// TIA Portal V17 export
// export: Created 2025-03-07T09:18:19.4347644Z, ExportSetting WithDefaults, DisplayName Totally Integrated Automation Portal, DisplayVersion V17 Update 8, DisplayName TIA Portal Openness, DisplayVersion V17 Update 8, DisplayName TIA Portal Version Control Interface, DisplayVersion V17, DisplayName SINAMICS Startdrive Advanced, DisplayVersion V17 SP2, DisplayName SINAMICS Startdrive G110M, G120, G120C, G120D, G120P, G115D, DisplayVersion V17 SP2, DisplayName SINAMICS Startdrive G130, G150, S120, S150, SINAMICS MV, S210, DisplayVersion V17 SP2, DisplayName STEP 7 Professional, DisplayVersion V17 Update 8, DisplayName SINUMERIK ONE STEP 7 Toolbox, DisplayVersion V17 Update 12, DisplayName SINUMERIK 840D sl STEP 7 Toolbox, DisplayVersion V17 Update 12, DisplayName STEP 7 Safety, DisplayVersion V17 Update 6, DisplayName WinCC Advanced, DisplayVersion V17 Update 8
FUNCTION "FC1702_ASPIRATION_VALVE" : Void   // FC1702, LAD
{ S7_Optimized_Access := 'TRUE' }
VERSION : 0.1
// stored: AutoNumber false, IsIECCheckEnabled false, SetENOAutomatically false, UDAEnableTagReadback false
BEGIN

REGION Network 1: <<<<<<<<<<<<<<<<<<<< ASPIRATION VALVES >>>>>>>>>>>>>>>>>>>>
END_REGION

REGION Network 2: <<<<<<<<<<<<<<<<<<<<<<<<<<< UNIT 01 >>>>>>>>>>>>>>>>>>>>>>>>>>>
END_REGION

REGION Network 3: CALL FB1701 UNIT 01 STATION 1 ASPIRATION ACTIVATION
   // 2#0000_0001 OPTIONS 0 BIT 0 SWITCHED ON INPUT 1 OPTION
   // 2#0000_0010 OPTIONS 0 BIT 1 SWITCHED ON INPUT 2 OPTION
   // 2#0000_0100 OPTIONS 0 BIT 2 SWITCHED ON INPUT 3 OPTION
   // 2#0000_1000 OPTIONS 0 BIT 3 SWITCHED ON INPUT 4 OPTION
   // 2#0001_0000 OPTIONS 0 BIT 4 SWITCHED OFF NOT SWITCHED ON INPUT 1 OPTION
   // 2#0010_0000 OPTIONS 0 BIT 5 SPARE
   // 2#0100_0000 OPTIONS 0 BIT 6 SPARE
   // 2#1000_0000 OPTIONS 0 BIT 7 SPARE
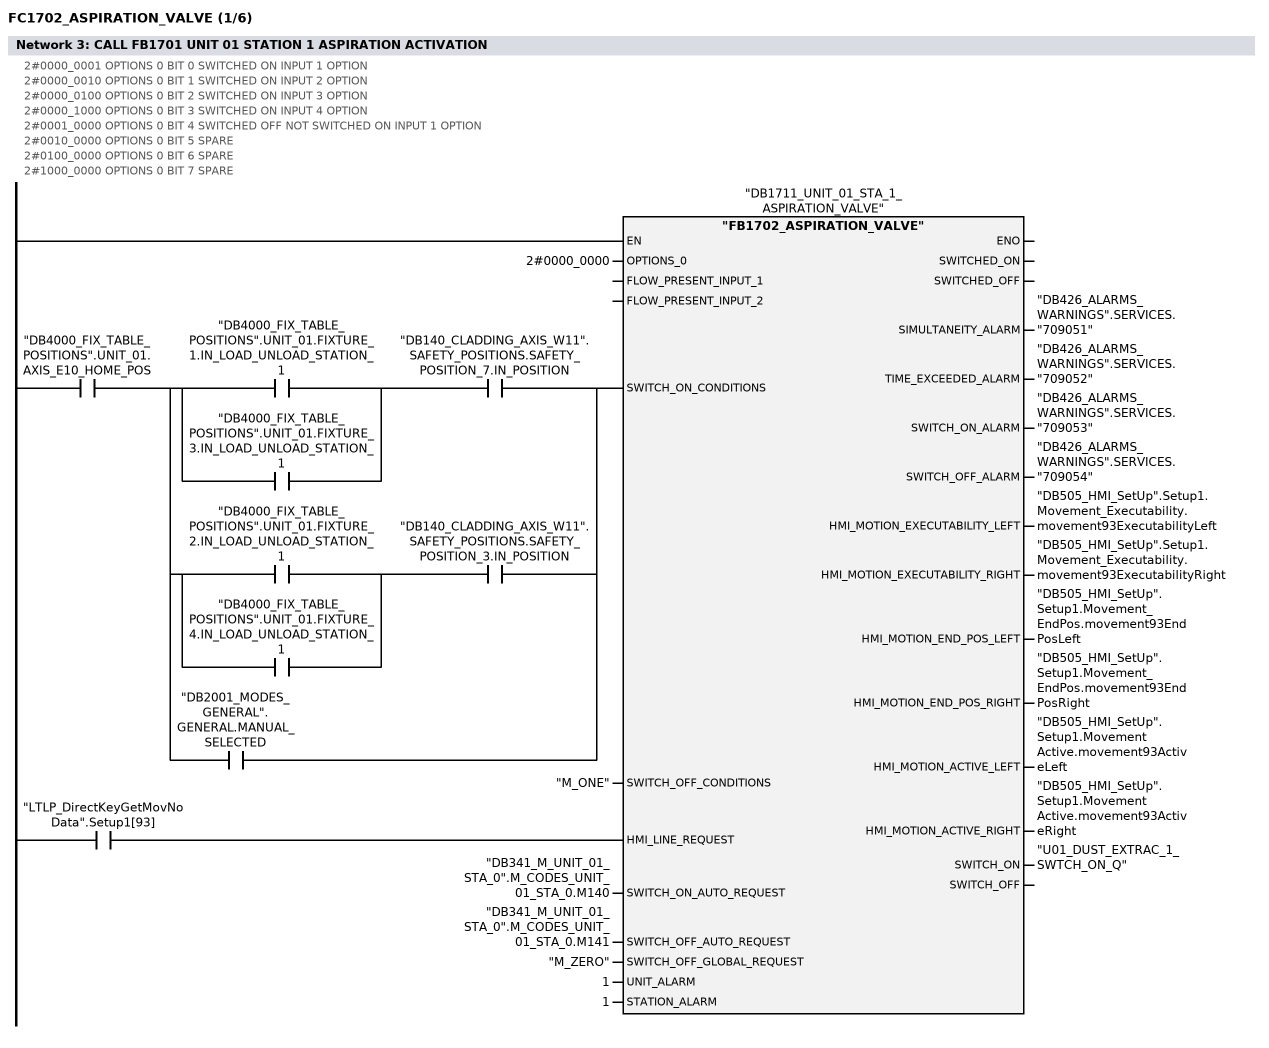
   RUNG wire#powerrail
      "DB1711_UNIT_01_STA_1_ASPIRATION_VALVE"(SWITCH_ON_CONDITIONS := wire#w4, HMI_LINE_REQUEST := wire#w5, OPTIONS_0 := 2#0000_0000, FLOW_PRESENT_INPUT_1 :=, FLOW_PRESENT_INPUT_2 :=, SWITCH_OFF_CONDITIONS := "M_ONE", SWITCH_ON_AUTO_REQUEST := "DB341_M_UNIT_01_STA_0".M_CODES_UNIT_01_STA_0.M140, SWITCH_OFF_AUTO_REQUEST := "DB341_M_UNIT_01_STA_0".M_CODES_UNIT_01_STA_0.M141, SWITCH_OFF_GLOBAL_REQUEST := "M_ZERO", UNIT_ALARM := 1, STATION_ALARM := 1, SWITCHED_ON =>, SWITCHED_OFF =>, SIMULTANEITY_ALARM => "DB426_ALARMS_WARNINGS".SERVICES."709051", TIME_EXCEEDED_ALARM => "DB426_ALARMS_WARNINGS".SERVICES."709052", SWITCH_ON_ALARM => "DB426_ALARMS_WARNINGS".SERVICES."709053", SWITCH_OFF_ALARM => "DB426_ALARMS_WARNINGS".SERVICES."709054", HMI_MOTION_EXECUTABILITY_LEFT => "DB505_HMI_SetUp".Setup1.Movement_Executability.movement93ExecutabilityLeft, HMI_MOTION_EXECUTABILITY_RIGHT => "DB505_HMI_SetUp".Setup1.Movement_Executability.movement93ExecutabilityRight, HMI_MOTION_END_POS_LEFT => "DB505_HMI_SetUp".Setup1.Movement_EndPos.movement93EndPosLeft, HMI_MOTION_END_POS_RIGHT => "DB505_HMI_SetUp".Setup1.Movement_EndPos.movement93EndPosRight, HMI_MOTION_ACTIVE_LEFT => "DB505_HMI_SetUp".Setup1.MovementActive.movement93ActiveLeft, HMI_MOTION_ACTIVE_RIGHT => "DB505_HMI_SetUp".Setup1.MovementActive.movement93ActiveRight, SWITCH_ON => "U01_DUST_EXTRAC_1_SWTCH_ON_Q", SWITCH_OFF =>)
   END_RUNG
   RUNG wire#powerrail
      Contact( "DB4000_FIX_TABLE_POSITIONS".UNIT_01.AXIS_E10_HOME_POS )
      wire#w1
      Contact( "DB4000_FIX_TABLE_POSITIONS".UNIT_01.FIXTURE_1.IN_LOAD_UNLOAD_STATION_1 )
      wire#w2
      Contact( "DB140_CLADDING_AXIS_W11".SAFETY_POSITIONS.SAFETY_POSITION_7.IN_POSITION )
   END_RUNG wire#w4
   RUNG wire#w1
      Contact( "DB4000_FIX_TABLE_POSITIONS".UNIT_01.FIXTURE_3.IN_LOAD_UNLOAD_STATION_1 )
   END_RUNG wire#w2
   RUNG wire#w1
      Contact( "DB4000_FIX_TABLE_POSITIONS".UNIT_01.FIXTURE_2.IN_LOAD_UNLOAD_STATION_1 )
      wire#w3
      Contact( "DB140_CLADDING_AXIS_W11".SAFETY_POSITIONS.SAFETY_POSITION_3.IN_POSITION )
   END_RUNG wire#w4
   RUNG wire#w1
      Contact( "DB4000_FIX_TABLE_POSITIONS".UNIT_01.FIXTURE_4.IN_LOAD_UNLOAD_STATION_1 )
   END_RUNG wire#w3
   RUNG wire#w1
      Contact( "DB2001_MODES_GENERAL".GENERAL.MANUAL_SELECTED )
   END_RUNG wire#w4
   RUNG wire#powerrail
      Contact( "LTLP_DirectKeyGetMovNoData".Setup1[93] )
   END_RUNG wire#w5
   // the same network as SCL:
   "DB1711_UNIT_01_STA_1_ASPIRATION_VALVE"(OPTIONS_0 := 2#0000_0000,   // "FB1702_ASPIRATION_VALVE"
                           SWITCH_ON_CONDITIONS := "DB4000_FIX_TABLE_POSITIONS".UNIT_01.AXIS_E10_HOME_POS AND ((("DB4000_FIX_TABLE_POSITIONS".UNIT_01.FIXTURE_1.IN_LOAD_UNLOAD_STATION_1 OR "DB4000_FIX_TABLE_POSITIONS".UNIT_01.FIXTURE_3.IN_LOAD_UNLOAD_STATION_1) AND "DB140_CLADDING_AXIS_W11".SAFETY_POSITIONS.SAFETY_POSITION_7.IN_POSITION) OR (("DB4000_FIX_TABLE_POSITIONS".UNIT_01.FIXTURE_2.IN_LOAD_UNLOAD_STATION_1 OR "DB4000_FIX_TABLE_POSITIONS".UNIT_01.FIXTURE_4.IN_LOAD_UNLOAD_STATION_1) AND "DB140_CLADDING_AXIS_W11".SAFETY_POSITIONS.SAFETY_POSITION_3.IN_POSITION) OR "DB2001_MODES_GENERAL".GENERAL.MANUAL_SELECTED),
                           SWITCH_OFF_CONDITIONS := "M_ONE",
                           HMI_LINE_REQUEST := "LTLP_DirectKeyGetMovNoData".Setup1[93],
                           SWITCH_ON_AUTO_REQUEST := "DB341_M_UNIT_01_STA_0".M_CODES_UNIT_01_STA_0.M140,
                           SWITCH_OFF_AUTO_REQUEST := "DB341_M_UNIT_01_STA_0".M_CODES_UNIT_01_STA_0.M141,
                           SWITCH_OFF_GLOBAL_REQUEST := "M_ZERO",
                           UNIT_ALARM := 1,
                           STATION_ALARM := 1,
                           SIMULTANEITY_ALARM => "DB426_ALARMS_WARNINGS".SERVICES."709051",
                           TIME_EXCEEDED_ALARM => "DB426_ALARMS_WARNINGS".SERVICES."709052",
                           SWITCH_ON_ALARM => "DB426_ALARMS_WARNINGS".SERVICES."709053",
                           SWITCH_OFF_ALARM => "DB426_ALARMS_WARNINGS".SERVICES."709054",
                           HMI_MOTION_EXECUTABILITY_LEFT => "DB505_HMI_SetUp".Setup1.Movement_Executability.movement93ExecutabilityLeft,
                           HMI_MOTION_EXECUTABILITY_RIGHT => "DB505_HMI_SetUp".Setup1.Movement_Executability.movement93ExecutabilityRight,
                           HMI_MOTION_END_POS_LEFT => "DB505_HMI_SetUp".Setup1.Movement_EndPos.movement93EndPosLeft,
                           HMI_MOTION_END_POS_RIGHT => "DB505_HMI_SetUp".Setup1.Movement_EndPos.movement93EndPosRight,
                           HMI_MOTION_ACTIVE_LEFT => "DB505_HMI_SetUp".Setup1.MovementActive.movement93ActiveLeft,
                           HMI_MOTION_ACTIVE_RIGHT => "DB505_HMI_SetUp".Setup1.MovementActive.movement93ActiveRight,
                           SWITCH_ON => "U01_DUST_EXTRAC_1_SWTCH_ON_Q");
END_REGION

REGION Network 4: CALL FB1701 UNIT 01 STATION 3 ASPIRATION ACTIVATION
   // 2#0000_0001 OPTIONS 0 BIT 0 SWITCHED ON INPUT 1 OPTION
   // 2#0000_0010 OPTIONS 0 BIT 1 SWITCHED ON INPUT 2 OPTION
   // 2#0000_0100 OPTIONS 0 BIT 2 SWITCHED ON INPUT 3 OPTION
   // 2#0000_1000 OPTIONS 0 BIT 3 SWITCHED ON INPUT 4 OPTION
   // 2#0001_0000 OPTIONS 0 BIT 4 SWITCHED OFF NOT SWITCHED ON INPUT 1 OPTION
   // 2#0010_0000 OPTIONS 0 BIT 5 SWITCHED ON WHEN CONTROL ON OPTION
   // 2#0100_0000 OPTIONS 0 BIT 6 SPARE
   // 2#1000_0000 OPTIONS 0 BIT 7 SPARE
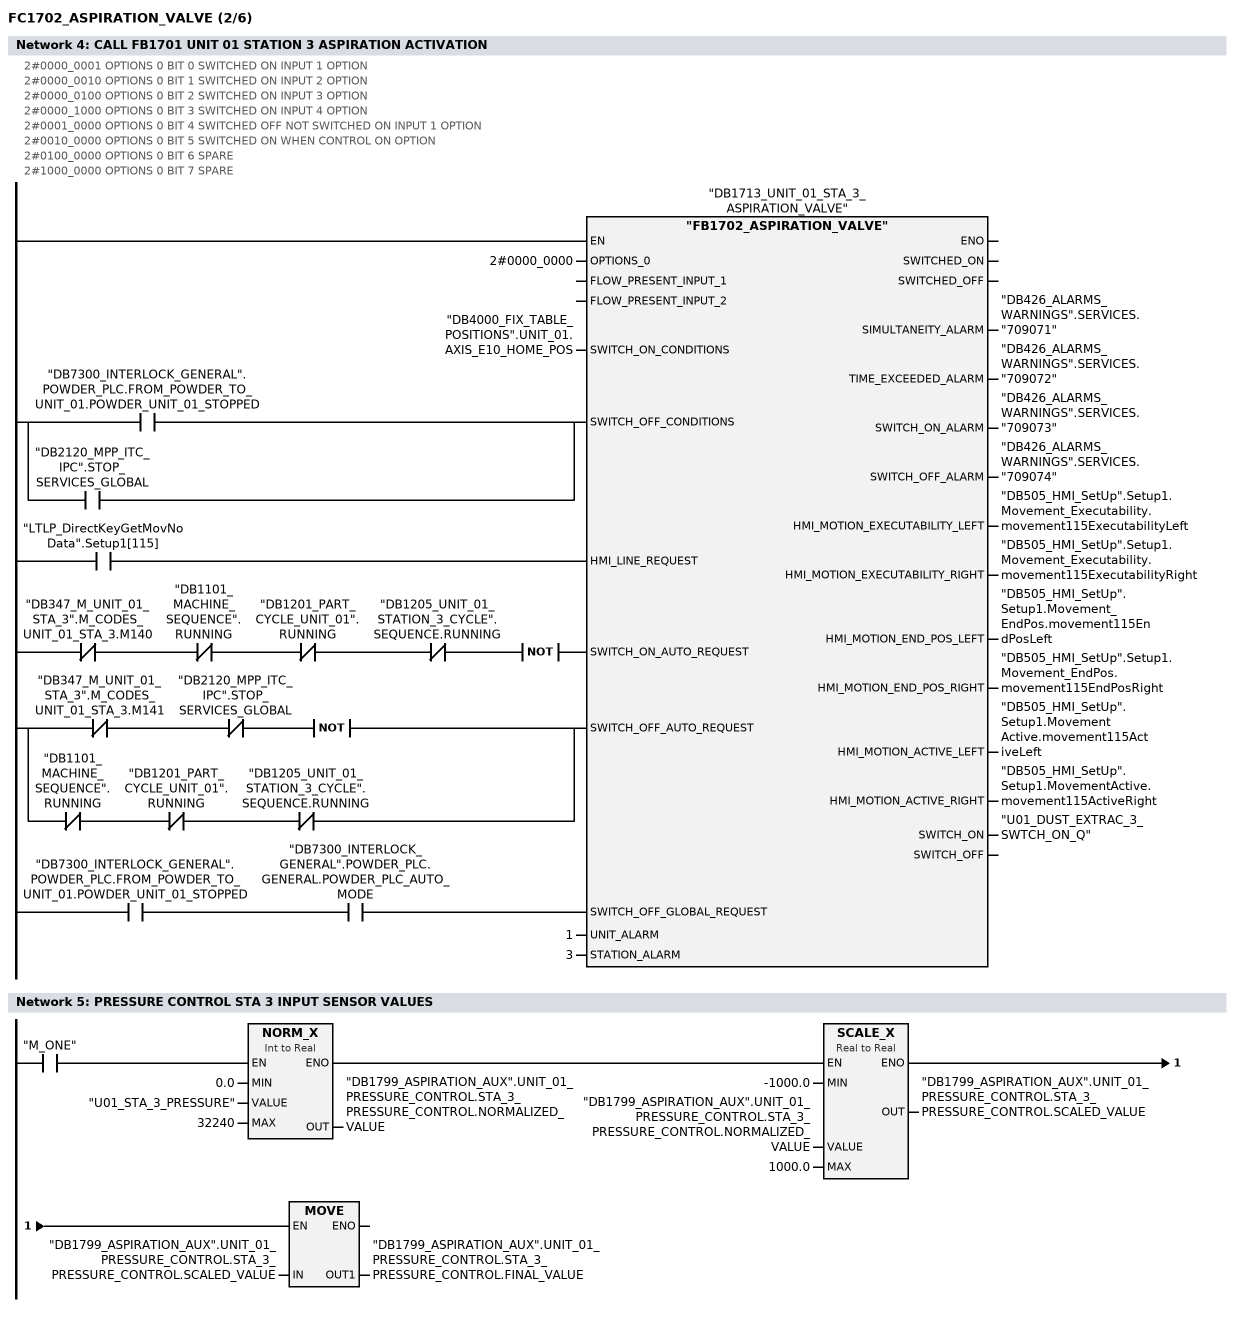
   RUNG wire#powerrail
      "DB1713_UNIT_01_STA_3_ASPIRATION_VALVE"(SWITCH_OFF_CONDITIONS := wire#w1, HMI_LINE_REQUEST := wire#w2, SWITCH_ON_AUTO_REQUEST := wire#w3, SWITCH_OFF_AUTO_REQUEST := wire#w4, SWITCH_OFF_GLOBAL_REQUEST := wire#w5, OPTIONS_0 := 2#0000_0000, FLOW_PRESENT_INPUT_1 :=, FLOW_PRESENT_INPUT_2 :=, SWITCH_ON_CONDITIONS := "DB4000_FIX_TABLE_POSITIONS".UNIT_01.AXIS_E10_HOME_POS, UNIT_ALARM := 1, STATION_ALARM := 3, SWITCHED_ON =>, SWITCHED_OFF =>, SIMULTANEITY_ALARM => "DB426_ALARMS_WARNINGS".SERVICES."709071", TIME_EXCEEDED_ALARM => "DB426_ALARMS_WARNINGS".SERVICES."709072", SWITCH_ON_ALARM => "DB426_ALARMS_WARNINGS".SERVICES."709073", SWITCH_OFF_ALARM => "DB426_ALARMS_WARNINGS".SERVICES."709074", HMI_MOTION_EXECUTABILITY_LEFT => "DB505_HMI_SetUp".Setup1.Movement_Executability.movement115ExecutabilityLeft, HMI_MOTION_EXECUTABILITY_RIGHT => "DB505_HMI_SetUp".Setup1.Movement_Executability.movement115ExecutabilityRight, HMI_MOTION_END_POS_LEFT => "DB505_HMI_SetUp".Setup1.Movement_EndPos.movement115EndPosLeft, HMI_MOTION_END_POS_RIGHT => "DB505_HMI_SetUp".Setup1.Movement_EndPos.movement115EndPosRight, HMI_MOTION_ACTIVE_LEFT => "DB505_HMI_SetUp".Setup1.MovementActive.movement115ActiveLeft, HMI_MOTION_ACTIVE_RIGHT => "DB505_HMI_SetUp".Setup1.MovementActive.movement115ActiveRight, SWITCH_ON => "U01_DUST_EXTRAC_3_SWTCH_ON_Q", SWITCH_OFF =>)
   END_RUNG
   RUNG wire#powerrail
      Contact( "DB7300_INTERLOCK_GENERAL".POWDER_PLC.FROM_POWDER_TO_UNIT_01.POWDER_UNIT_01_STOPPED )
   END_RUNG wire#w1
   RUNG wire#powerrail
      Contact( "DB2120_MPP_ITC_IPC".STOP_SERVICES_GLOBAL )
   END_RUNG wire#w1
   RUNG wire#powerrail
      Contact( "LTLP_DirectKeyGetMovNoData".Setup1[115] )
   END_RUNG wire#w2
   RUNG wire#powerrail
      I_Contact( "DB347_M_UNIT_01_STA_3".M_CODES_UNIT_01_STA_3.M140 )
      I_Contact( "DB1101_MACHINE_SEQUENCE".RUNNING )
      I_Contact( "DB1201_PART_CYCLE_UNIT_01".RUNNING )
      I_Contact( "DB1205_UNIT_01_STATION_3_CYCLE".SEQUENCE.RUNNING )
      Not()
   END_RUNG wire#w3
   RUNG wire#powerrail
      I_Contact( "DB347_M_UNIT_01_STA_3".M_CODES_UNIT_01_STA_3.M141 )
      I_Contact( "DB2120_MPP_ITC_IPC".STOP_SERVICES_GLOBAL )
      Not()
   END_RUNG wire#w4
   RUNG wire#powerrail
      I_Contact( "DB1101_MACHINE_SEQUENCE".RUNNING )
      I_Contact( "DB1201_PART_CYCLE_UNIT_01".RUNNING )
      I_Contact( "DB1205_UNIT_01_STATION_3_CYCLE".SEQUENCE.RUNNING )
   END_RUNG wire#w4
   RUNG wire#powerrail
      Contact( "DB7300_INTERLOCK_GENERAL".POWDER_PLC.FROM_POWDER_TO_UNIT_01.POWDER_UNIT_01_STOPPED )
      Contact( "DB7300_INTERLOCK_GENERAL".POWDER_PLC.GENERAL.POWDER_PLC_AUTO_MODE )
   END_RUNG wire#w5
   // the same network as SCL:
   "DB1713_UNIT_01_STA_3_ASPIRATION_VALVE"(OPTIONS_0 := 2#0000_0000,   // "FB1702_ASPIRATION_VALVE"
                           SWITCH_ON_CONDITIONS := "DB4000_FIX_TABLE_POSITIONS".UNIT_01.AXIS_E10_HOME_POS,
                           SWITCH_OFF_CONDITIONS := "DB7300_INTERLOCK_GENERAL".POWDER_PLC.FROM_POWDER_TO_UNIT_01.POWDER_UNIT_01_STOPPED OR "DB2120_MPP_ITC_IPC".STOP_SERVICES_GLOBAL,
                           HMI_LINE_REQUEST := "LTLP_DirectKeyGetMovNoData".Setup1[115],
                           SWITCH_ON_AUTO_REQUEST := NOT (NOT "DB347_M_UNIT_01_STA_3".M_CODES_UNIT_01_STA_3.M140 AND NOT "DB1101_MACHINE_SEQUENCE".RUNNING AND NOT "DB1201_PART_CYCLE_UNIT_01".RUNNING AND NOT "DB1205_UNIT_01_STATION_3_CYCLE".SEQUENCE.RUNNING),
                           SWITCH_OFF_AUTO_REQUEST := NOT (NOT "DB347_M_UNIT_01_STA_3".M_CODES_UNIT_01_STA_3.M141 AND NOT "DB2120_MPP_ITC_IPC".STOP_SERVICES_GLOBAL) OR (NOT "DB1101_MACHINE_SEQUENCE".RUNNING AND NOT "DB1201_PART_CYCLE_UNIT_01".RUNNING AND NOT "DB1205_UNIT_01_STATION_3_CYCLE".SEQUENCE.RUNNING),
                           SWITCH_OFF_GLOBAL_REQUEST := "DB7300_INTERLOCK_GENERAL".POWDER_PLC.FROM_POWDER_TO_UNIT_01.POWDER_UNIT_01_STOPPED AND "DB7300_INTERLOCK_GENERAL".POWDER_PLC.GENERAL.POWDER_PLC_AUTO_MODE,
                           UNIT_ALARM := 1,
                           STATION_ALARM := 3,
                           SIMULTANEITY_ALARM => "DB426_ALARMS_WARNINGS".SERVICES."709071",
                           TIME_EXCEEDED_ALARM => "DB426_ALARMS_WARNINGS".SERVICES."709072",
                           SWITCH_ON_ALARM => "DB426_ALARMS_WARNINGS".SERVICES."709073",
                           SWITCH_OFF_ALARM => "DB426_ALARMS_WARNINGS".SERVICES."709074",
                           HMI_MOTION_EXECUTABILITY_LEFT => "DB505_HMI_SetUp".Setup1.Movement_Executability.movement115ExecutabilityLeft,
                           HMI_MOTION_EXECUTABILITY_RIGHT => "DB505_HMI_SetUp".Setup1.Movement_Executability.movement115ExecutabilityRight,
                           HMI_MOTION_END_POS_LEFT => "DB505_HMI_SetUp".Setup1.Movement_EndPos.movement115EndPosLeft,
                           HMI_MOTION_END_POS_RIGHT => "DB505_HMI_SetUp".Setup1.Movement_EndPos.movement115EndPosRight,
                           HMI_MOTION_ACTIVE_LEFT => "DB505_HMI_SetUp".Setup1.MovementActive.movement115ActiveLeft,
                           HMI_MOTION_ACTIVE_RIGHT => "DB505_HMI_SetUp".Setup1.MovementActive.movement115ActiveRight,
                           SWITCH_ON => "U01_DUST_EXTRAC_3_SWTCH_ON_Q");
END_REGION

REGION Network 5: PRESSURE CONTROL STA 3 INPUT SENSOR VALUES
   RUNG wire#powerrail
      Contact( "M_ONE" )
      { S7_Templates := "[SrcType := Int, DestType := Real]" } Normalize(min := 0.0, value := "U01_STA_3_PRESSURE", max := 32240, out => "DB1799_ASPIRATION_AUX".UNIT_01_PRESSURE_CONTROL.STA_3_PRESSURE_CONTROL.NORMALIZED_VALUE)
      { S7_Templates := "[SrcType := Real, DestType := Real]" } Scale(min := -1000.0, value := "DB1799_ASPIRATION_AUX".UNIT_01_PRESSURE_CONTROL.STA_3_PRESSURE_CONTROL.NORMALIZED_VALUE, max := 1000.0, out => "DB1799_ASPIRATION_AUX".UNIT_01_PRESSURE_CONTROL.STA_3_PRESSURE_CONTROL.SCALED_VALUE)
      Move(in := "DB1799_ASPIRATION_AUX".UNIT_01_PRESSURE_CONTROL.STA_3_PRESSURE_CONTROL.SCALED_VALUE, out1 => "DB1799_ASPIRATION_AUX".UNIT_01_PRESSURE_CONTROL.STA_3_PRESSURE_CONTROL.FINAL_VALUE)
   END_RUNG
   // the same network as SCL:
   IF "M_ONE" THEN
       "DB1799_ASPIRATION_AUX".UNIT_01_PRESSURE_CONTROL.STA_3_PRESSURE_CONTROL.NORMALIZED_VALUE := NORM_X(MIN := 0.0, VALUE := "U01_STA_3_PRESSURE", MAX := 32240);
       "DB1799_ASPIRATION_AUX".UNIT_01_PRESSURE_CONTROL.STA_3_PRESSURE_CONTROL.SCALED_VALUE := SCALE_X(MIN := -1000.0, VALUE := "DB1799_ASPIRATION_AUX".UNIT_01_PRESSURE_CONTROL.STA_3_PRESSURE_CONTROL.NORMALIZED_VALUE, MAX := 1000.0);
       "DB1799_ASPIRATION_AUX".UNIT_01_PRESSURE_CONTROL.STA_3_PRESSURE_CONTROL.FINAL_VALUE := "DB1799_ASPIRATION_AUX".UNIT_01_PRESSURE_CONTROL.STA_3_PRESSURE_CONTROL.SCALED_VALUE;
   END_IF;
END_REGION

REGION Network 6: CALL FB1701 UNIT 01 STATION 4 ASPIRATION ACTIVATION
   // 2#0000_0001 OPTIONS 0 BIT 0 SWITCHED ON INPUT 1 OPTION
   // 2#0000_0010 OPTIONS 0 BIT 1 SWITCHED ON INPUT 2 OPTION
   // 2#0000_0100 OPTIONS 0 BIT 2 SWITCHED ON INPUT 3 OPTION
   // 2#0000_1000 OPTIONS 0 BIT 3 SWITCHED ON INPUT 4 OPTION
   // 2#0001_0000 OPTIONS 0 BIT 4 SWITCHED OFF NOT SWITCHED ON INPUT 1 OPTION
   // 2#0010_0000 OPTIONS 0 BIT 5 SPARE
   // 2#0100_0000 OPTIONS 0 BIT 6 SPARE
   // 2#1000_0000 OPTIONS 0 BIT 7 SPARE
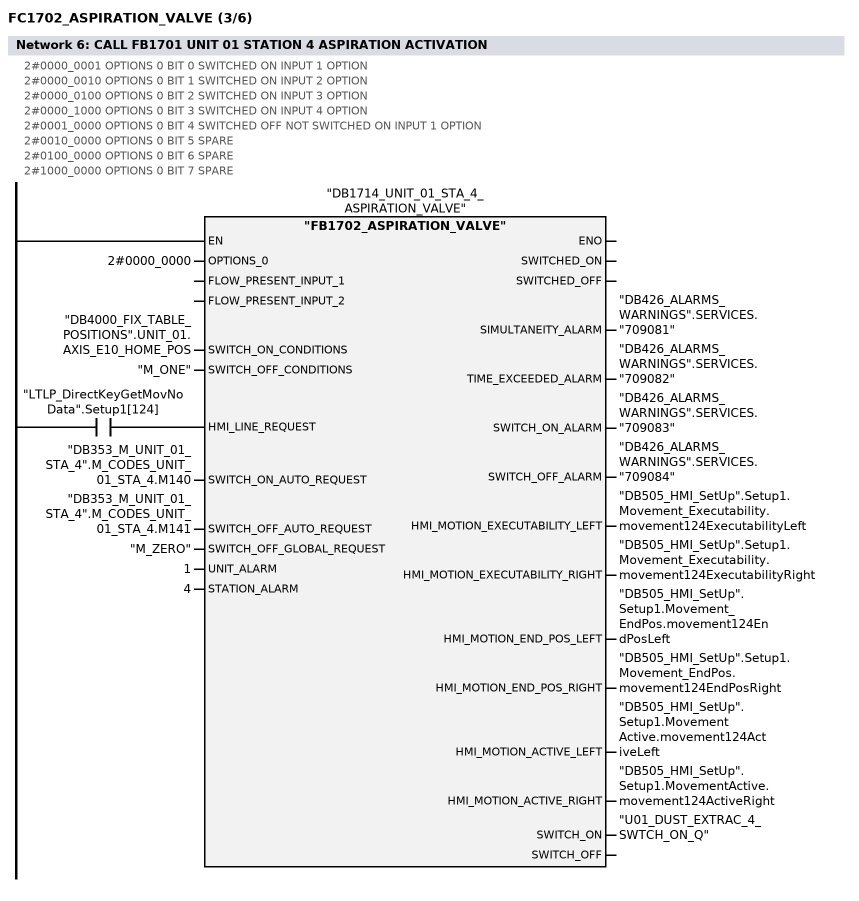
   RUNG wire#powerrail
      "DB1714_UNIT_01_STA_4_ASPIRATION_VALVE"(HMI_LINE_REQUEST := wire#w1, OPTIONS_0 := 2#0000_0000, FLOW_PRESENT_INPUT_1 :=, FLOW_PRESENT_INPUT_2 :=, SWITCH_ON_CONDITIONS := "DB4000_FIX_TABLE_POSITIONS".UNIT_01.AXIS_E10_HOME_POS, SWITCH_OFF_CONDITIONS := "M_ONE", SWITCH_ON_AUTO_REQUEST := "DB353_M_UNIT_01_STA_4".M_CODES_UNIT_01_STA_4.M140, SWITCH_OFF_AUTO_REQUEST := "DB353_M_UNIT_01_STA_4".M_CODES_UNIT_01_STA_4.M141, SWITCH_OFF_GLOBAL_REQUEST := "M_ZERO", UNIT_ALARM := 1, STATION_ALARM := 4, SWITCHED_ON =>, SWITCHED_OFF =>, SIMULTANEITY_ALARM => "DB426_ALARMS_WARNINGS".SERVICES."709081", TIME_EXCEEDED_ALARM => "DB426_ALARMS_WARNINGS".SERVICES."709082", SWITCH_ON_ALARM => "DB426_ALARMS_WARNINGS".SERVICES."709083", SWITCH_OFF_ALARM => "DB426_ALARMS_WARNINGS".SERVICES."709084", HMI_MOTION_EXECUTABILITY_LEFT => "DB505_HMI_SetUp".Setup1.Movement_Executability.movement124ExecutabilityLeft, HMI_MOTION_EXECUTABILITY_RIGHT => "DB505_HMI_SetUp".Setup1.Movement_Executability.movement124ExecutabilityRight, HMI_MOTION_END_POS_LEFT => "DB505_HMI_SetUp".Setup1.Movement_EndPos.movement124EndPosLeft, HMI_MOTION_END_POS_RIGHT => "DB505_HMI_SetUp".Setup1.Movement_EndPos.movement124EndPosRight, HMI_MOTION_ACTIVE_LEFT => "DB505_HMI_SetUp".Setup1.MovementActive.movement124ActiveLeft, HMI_MOTION_ACTIVE_RIGHT => "DB505_HMI_SetUp".Setup1.MovementActive.movement124ActiveRight, SWITCH_ON => "U01_DUST_EXTRAC_4_SWTCH_ON_Q", SWITCH_OFF =>)
   END_RUNG
   RUNG wire#powerrail
      Contact( "LTLP_DirectKeyGetMovNoData".Setup1[124] )
   END_RUNG wire#w1
   // the same network as SCL:
   "DB1714_UNIT_01_STA_4_ASPIRATION_VALVE"(OPTIONS_0 := 2#0000_0000,   // "FB1702_ASPIRATION_VALVE"
                           SWITCH_ON_CONDITIONS := "DB4000_FIX_TABLE_POSITIONS".UNIT_01.AXIS_E10_HOME_POS,
                           SWITCH_OFF_CONDITIONS := "M_ONE",
                           HMI_LINE_REQUEST := "LTLP_DirectKeyGetMovNoData".Setup1[124],
                           SWITCH_ON_AUTO_REQUEST := "DB353_M_UNIT_01_STA_4".M_CODES_UNIT_01_STA_4.M140,
                           SWITCH_OFF_AUTO_REQUEST := "DB353_M_UNIT_01_STA_4".M_CODES_UNIT_01_STA_4.M141,
                           SWITCH_OFF_GLOBAL_REQUEST := "M_ZERO",
                           UNIT_ALARM := 1,
                           STATION_ALARM := 4,
                           SIMULTANEITY_ALARM => "DB426_ALARMS_WARNINGS".SERVICES."709081",
                           TIME_EXCEEDED_ALARM => "DB426_ALARMS_WARNINGS".SERVICES."709082",
                           SWITCH_ON_ALARM => "DB426_ALARMS_WARNINGS".SERVICES."709083",
                           SWITCH_OFF_ALARM => "DB426_ALARMS_WARNINGS".SERVICES."709084",
                           HMI_MOTION_EXECUTABILITY_LEFT => "DB505_HMI_SetUp".Setup1.Movement_Executability.movement124ExecutabilityLeft,
                           HMI_MOTION_EXECUTABILITY_RIGHT => "DB505_HMI_SetUp".Setup1.Movement_Executability.movement124ExecutabilityRight,
                           HMI_MOTION_END_POS_LEFT => "DB505_HMI_SetUp".Setup1.Movement_EndPos.movement124EndPosLeft,
                           HMI_MOTION_END_POS_RIGHT => "DB505_HMI_SetUp".Setup1.Movement_EndPos.movement124EndPosRight,
                           HMI_MOTION_ACTIVE_LEFT => "DB505_HMI_SetUp".Setup1.MovementActive.movement124ActiveLeft,
                           HMI_MOTION_ACTIVE_RIGHT => "DB505_HMI_SetUp".Setup1.MovementActive.movement124ActiveRight,
                           SWITCH_ON => "U01_DUST_EXTRAC_4_SWTCH_ON_Q");
END_REGION

REGION Network 7: <<<<<<<<<<<<<<<<<<<<<<<<<<< UNIT 02 >>>>>>>>>>>>>>>>>>>>>>>>>>>
END_REGION

REGION Network 8: CALL FB1701 UNIT 02 STATION 1 ASPIRATION ACTIVATION
   // 2#0000_0001 OPTIONS 0 BIT 0 SWITCHED ON INPUT 1 OPTION
   // 2#0000_0010 OPTIONS 0 BIT 1 SWITCHED ON INPUT 2 OPTION
   // 2#0000_0100 OPTIONS 0 BIT 2 SWITCHED ON INPUT 3 OPTION
   // 2#0000_1000 OPTIONS 0 BIT 3 SWITCHED ON INPUT 4 OPTION
   // 2#0001_0000 OPTIONS 0 BIT 4 SWITCHED OFF NOT SWITCHED ON INPUT 1 OPTION
   // 2#0010_0000 OPTIONS 0 BIT 5 SPARE
   // 2#0100_0000 OPTIONS 0 BIT 6 SPARE
   // 2#1000_0000 OPTIONS 0 BIT 7 SPARE
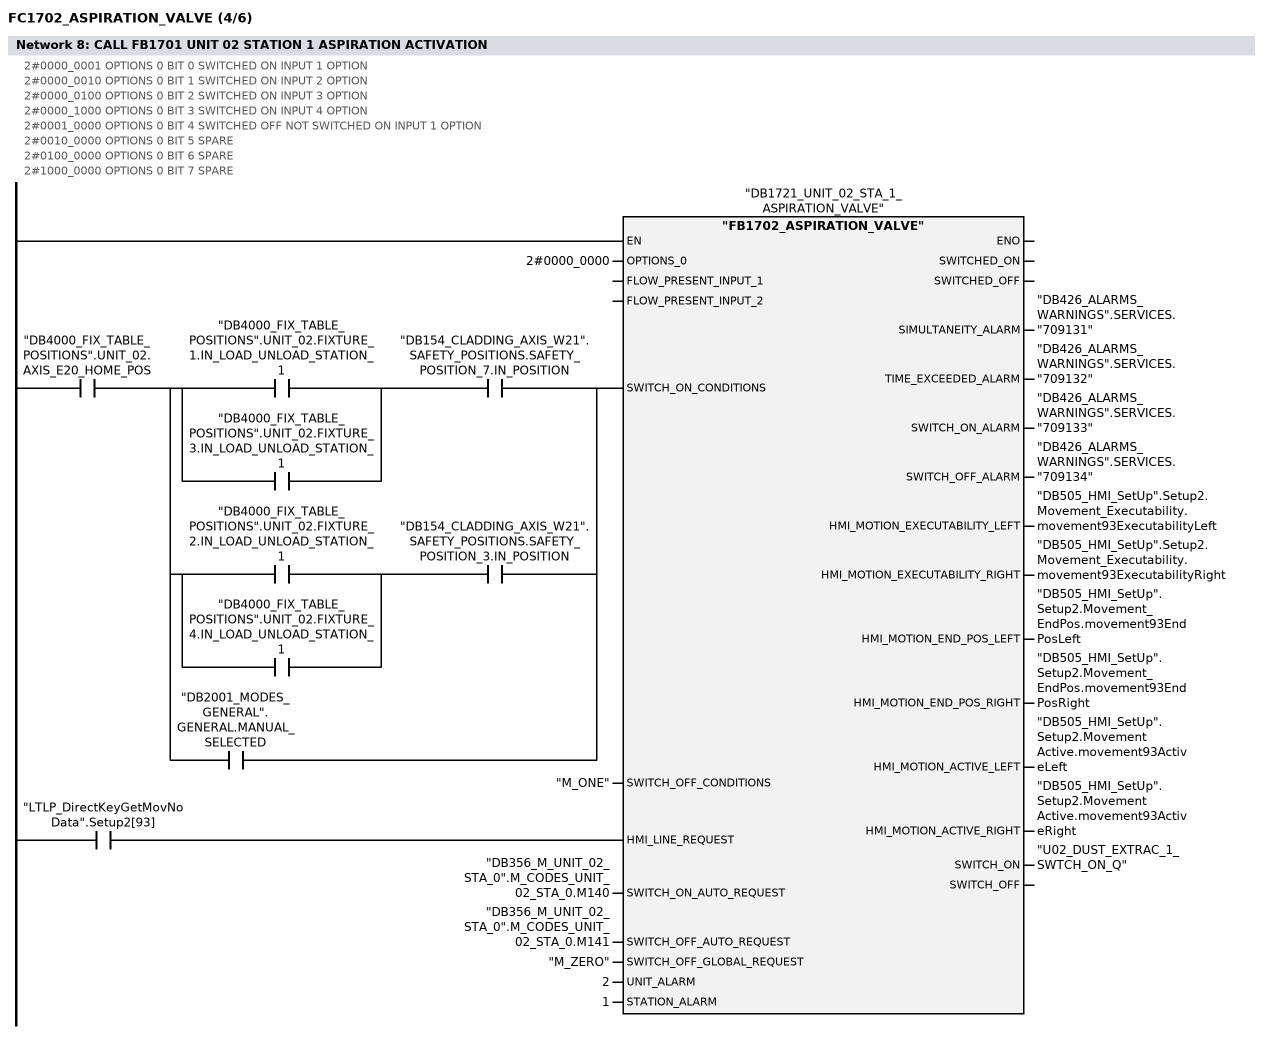
   RUNG wire#powerrail
      "DB1721_UNIT_02_STA_1_ASPIRATION_VALVE"(SWITCH_ON_CONDITIONS := wire#w4, HMI_LINE_REQUEST := wire#w5, OPTIONS_0 := 2#0000_0000, FLOW_PRESENT_INPUT_1 :=, FLOW_PRESENT_INPUT_2 :=, SWITCH_OFF_CONDITIONS := "M_ONE", SWITCH_ON_AUTO_REQUEST := "DB356_M_UNIT_02_STA_0".M_CODES_UNIT_02_STA_0.M140, SWITCH_OFF_AUTO_REQUEST := "DB356_M_UNIT_02_STA_0".M_CODES_UNIT_02_STA_0.M141, SWITCH_OFF_GLOBAL_REQUEST := "M_ZERO", UNIT_ALARM := 2, STATION_ALARM := 1, SWITCHED_ON =>, SWITCHED_OFF =>, SIMULTANEITY_ALARM => "DB426_ALARMS_WARNINGS".SERVICES."709131", TIME_EXCEEDED_ALARM => "DB426_ALARMS_WARNINGS".SERVICES."709132", SWITCH_ON_ALARM => "DB426_ALARMS_WARNINGS".SERVICES."709133", SWITCH_OFF_ALARM => "DB426_ALARMS_WARNINGS".SERVICES."709134", HMI_MOTION_EXECUTABILITY_LEFT => "DB505_HMI_SetUp".Setup2.Movement_Executability.movement93ExecutabilityLeft, HMI_MOTION_EXECUTABILITY_RIGHT => "DB505_HMI_SetUp".Setup2.Movement_Executability.movement93ExecutabilityRight, HMI_MOTION_END_POS_LEFT => "DB505_HMI_SetUp".Setup2.Movement_EndPos.movement93EndPosLeft, HMI_MOTION_END_POS_RIGHT => "DB505_HMI_SetUp".Setup2.Movement_EndPos.movement93EndPosRight, HMI_MOTION_ACTIVE_LEFT => "DB505_HMI_SetUp".Setup2.MovementActive.movement93ActiveLeft, HMI_MOTION_ACTIVE_RIGHT => "DB505_HMI_SetUp".Setup2.MovementActive.movement93ActiveRight, SWITCH_ON => "U02_DUST_EXTRAC_1_SWTCH_ON_Q", SWITCH_OFF =>)
   END_RUNG
   RUNG wire#powerrail
      Contact( "DB4000_FIX_TABLE_POSITIONS".UNIT_02.AXIS_E20_HOME_POS )
      wire#w1
      Contact( "DB4000_FIX_TABLE_POSITIONS".UNIT_02.FIXTURE_1.IN_LOAD_UNLOAD_STATION_1 )
      wire#w2
      Contact( "DB154_CLADDING_AXIS_W21".SAFETY_POSITIONS.SAFETY_POSITION_7.IN_POSITION )
   END_RUNG wire#w4
   RUNG wire#w1
      Contact( "DB4000_FIX_TABLE_POSITIONS".UNIT_02.FIXTURE_3.IN_LOAD_UNLOAD_STATION_1 )
   END_RUNG wire#w2
   RUNG wire#w1
      Contact( "DB4000_FIX_TABLE_POSITIONS".UNIT_02.FIXTURE_2.IN_LOAD_UNLOAD_STATION_1 )
      wire#w3
      Contact( "DB154_CLADDING_AXIS_W21".SAFETY_POSITIONS.SAFETY_POSITION_3.IN_POSITION )
   END_RUNG wire#w4
   RUNG wire#w1
      Contact( "DB4000_FIX_TABLE_POSITIONS".UNIT_02.FIXTURE_4.IN_LOAD_UNLOAD_STATION_1 )
   END_RUNG wire#w3
   RUNG wire#w1
      Contact( "DB2001_MODES_GENERAL".GENERAL.MANUAL_SELECTED )
   END_RUNG wire#w4
   RUNG wire#powerrail
      Contact( "LTLP_DirectKeyGetMovNoData".Setup2[93] )
   END_RUNG wire#w5
   // the same network as SCL:
   "DB1721_UNIT_02_STA_1_ASPIRATION_VALVE"(OPTIONS_0 := 2#0000_0000,   // "FB1702_ASPIRATION_VALVE"
                           SWITCH_ON_CONDITIONS := "DB4000_FIX_TABLE_POSITIONS".UNIT_02.AXIS_E20_HOME_POS AND ((("DB4000_FIX_TABLE_POSITIONS".UNIT_02.FIXTURE_1.IN_LOAD_UNLOAD_STATION_1 OR "DB4000_FIX_TABLE_POSITIONS".UNIT_02.FIXTURE_3.IN_LOAD_UNLOAD_STATION_1) AND "DB154_CLADDING_AXIS_W21".SAFETY_POSITIONS.SAFETY_POSITION_7.IN_POSITION) OR (("DB4000_FIX_TABLE_POSITIONS".UNIT_02.FIXTURE_2.IN_LOAD_UNLOAD_STATION_1 OR "DB4000_FIX_TABLE_POSITIONS".UNIT_02.FIXTURE_4.IN_LOAD_UNLOAD_STATION_1) AND "DB154_CLADDING_AXIS_W21".SAFETY_POSITIONS.SAFETY_POSITION_3.IN_POSITION) OR "DB2001_MODES_GENERAL".GENERAL.MANUAL_SELECTED),
                           SWITCH_OFF_CONDITIONS := "M_ONE",
                           HMI_LINE_REQUEST := "LTLP_DirectKeyGetMovNoData".Setup2[93],
                           SWITCH_ON_AUTO_REQUEST := "DB356_M_UNIT_02_STA_0".M_CODES_UNIT_02_STA_0.M140,
                           SWITCH_OFF_AUTO_REQUEST := "DB356_M_UNIT_02_STA_0".M_CODES_UNIT_02_STA_0.M141,
                           SWITCH_OFF_GLOBAL_REQUEST := "M_ZERO",
                           UNIT_ALARM := 2,
                           STATION_ALARM := 1,
                           SIMULTANEITY_ALARM => "DB426_ALARMS_WARNINGS".SERVICES."709131",
                           TIME_EXCEEDED_ALARM => "DB426_ALARMS_WARNINGS".SERVICES."709132",
                           SWITCH_ON_ALARM => "DB426_ALARMS_WARNINGS".SERVICES."709133",
                           SWITCH_OFF_ALARM => "DB426_ALARMS_WARNINGS".SERVICES."709134",
                           HMI_MOTION_EXECUTABILITY_LEFT => "DB505_HMI_SetUp".Setup2.Movement_Executability.movement93ExecutabilityLeft,
                           HMI_MOTION_EXECUTABILITY_RIGHT => "DB505_HMI_SetUp".Setup2.Movement_Executability.movement93ExecutabilityRight,
                           HMI_MOTION_END_POS_LEFT => "DB505_HMI_SetUp".Setup2.Movement_EndPos.movement93EndPosLeft,
                           HMI_MOTION_END_POS_RIGHT => "DB505_HMI_SetUp".Setup2.Movement_EndPos.movement93EndPosRight,
                           HMI_MOTION_ACTIVE_LEFT => "DB505_HMI_SetUp".Setup2.MovementActive.movement93ActiveLeft,
                           HMI_MOTION_ACTIVE_RIGHT => "DB505_HMI_SetUp".Setup2.MovementActive.movement93ActiveRight,
                           SWITCH_ON => "U02_DUST_EXTRAC_1_SWTCH_ON_Q");
END_REGION

REGION Network 9: CALL FB1701 UNIT 02 STATION 3 ASPIRATION ACTIVATION
   // 2#0000_0001 OPTIONS 0 BIT 0 SWITCHED ON INPUT 1 OPTION
   // 2#0000_0010 OPTIONS 0 BIT 1 SWITCHED ON INPUT 2 OPTION
   // 2#0000_0100 OPTIONS 0 BIT 2 SWITCHED ON INPUT 3 OPTION
   // 2#0000_1000 OPTIONS 0 BIT 3 SWITCHED ON INPUT 4 OPTION
   // 2#0001_0000 OPTIONS 0 BIT 4 SWITCHED OFF NOT SWITCHED ON INPUT 1 OPTION
   // 2#0010_0000 OPTIONS 0 BIT 5 SWITCHED ON WHEN CONTROL ON OPTION
   // 2#0100_0000 OPTIONS 0 BIT 6 SPARE
   // 2#1000_0000 OPTIONS 0 BIT 7 SPARE
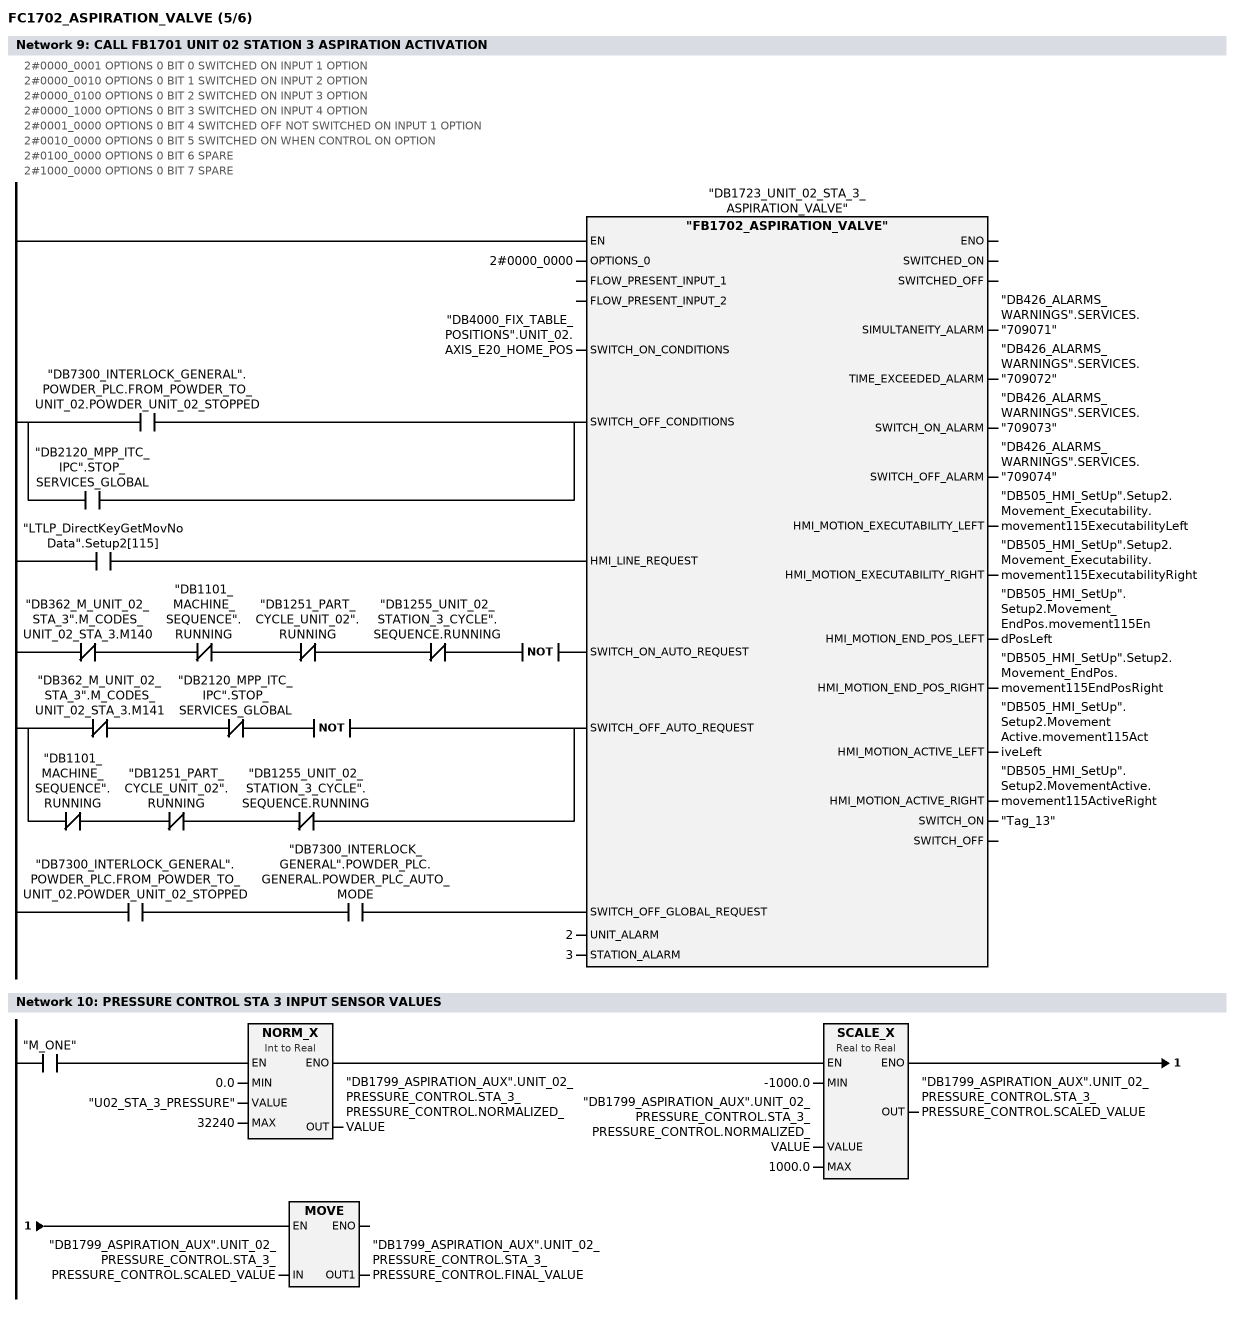
   RUNG wire#powerrail
      "DB1723_UNIT_02_STA_3_ASPIRATION_VALVE"(SWITCH_OFF_CONDITIONS := wire#w1, HMI_LINE_REQUEST := wire#w2, SWITCH_ON_AUTO_REQUEST := wire#w3, SWITCH_OFF_AUTO_REQUEST := wire#w4, SWITCH_OFF_GLOBAL_REQUEST := wire#w5, OPTIONS_0 := 2#0000_0000, FLOW_PRESENT_INPUT_1 :=, FLOW_PRESENT_INPUT_2 :=, SWITCH_ON_CONDITIONS := "DB4000_FIX_TABLE_POSITIONS".UNIT_02.AXIS_E20_HOME_POS, UNIT_ALARM := 2, STATION_ALARM := 3, SWITCHED_ON =>, SWITCHED_OFF =>, SIMULTANEITY_ALARM => "DB426_ALARMS_WARNINGS".SERVICES."709071", TIME_EXCEEDED_ALARM => "DB426_ALARMS_WARNINGS".SERVICES."709072", SWITCH_ON_ALARM => "DB426_ALARMS_WARNINGS".SERVICES."709073", SWITCH_OFF_ALARM => "DB426_ALARMS_WARNINGS".SERVICES."709074", HMI_MOTION_EXECUTABILITY_LEFT => "DB505_HMI_SetUp".Setup2.Movement_Executability.movement115ExecutabilityLeft, HMI_MOTION_EXECUTABILITY_RIGHT => "DB505_HMI_SetUp".Setup2.Movement_Executability.movement115ExecutabilityRight, HMI_MOTION_END_POS_LEFT => "DB505_HMI_SetUp".Setup2.Movement_EndPos.movement115EndPosLeft, HMI_MOTION_END_POS_RIGHT => "DB505_HMI_SetUp".Setup2.Movement_EndPos.movement115EndPosRight, HMI_MOTION_ACTIVE_LEFT => "DB505_HMI_SetUp".Setup2.MovementActive.movement115ActiveLeft, HMI_MOTION_ACTIVE_RIGHT => "DB505_HMI_SetUp".Setup2.MovementActive.movement115ActiveRight, SWITCH_ON => "Tag_13", SWITCH_OFF =>)
   END_RUNG
   RUNG wire#powerrail
      Contact( "DB7300_INTERLOCK_GENERAL".POWDER_PLC.FROM_POWDER_TO_UNIT_02.POWDER_UNIT_02_STOPPED )
   END_RUNG wire#w1
   RUNG wire#powerrail
      Contact( "DB2120_MPP_ITC_IPC".STOP_SERVICES_GLOBAL )
   END_RUNG wire#w1
   RUNG wire#powerrail
      Contact( "LTLP_DirectKeyGetMovNoData".Setup2[115] )
   END_RUNG wire#w2
   RUNG wire#powerrail
      I_Contact( "DB362_M_UNIT_02_STA_3".M_CODES_UNIT_02_STA_3.M140 )
      I_Contact( "DB1101_MACHINE_SEQUENCE".RUNNING )
      I_Contact( "DB1251_PART_CYCLE_UNIT_02".RUNNING )
      I_Contact( "DB1255_UNIT_02_STATION_3_CYCLE".SEQUENCE.RUNNING )
      Not()
   END_RUNG wire#w3
   RUNG wire#powerrail
      I_Contact( "DB362_M_UNIT_02_STA_3".M_CODES_UNIT_02_STA_3.M141 )
      I_Contact( "DB2120_MPP_ITC_IPC".STOP_SERVICES_GLOBAL )
      Not()
   END_RUNG wire#w4
   RUNG wire#powerrail
      I_Contact( "DB1101_MACHINE_SEQUENCE".RUNNING )
      I_Contact( "DB1251_PART_CYCLE_UNIT_02".RUNNING )
      I_Contact( "DB1255_UNIT_02_STATION_3_CYCLE".SEQUENCE.RUNNING )
   END_RUNG wire#w4
   RUNG wire#powerrail
      Contact( "DB7300_INTERLOCK_GENERAL".POWDER_PLC.FROM_POWDER_TO_UNIT_02.POWDER_UNIT_02_STOPPED )
      Contact( "DB7300_INTERLOCK_GENERAL".POWDER_PLC.GENERAL.POWDER_PLC_AUTO_MODE )
   END_RUNG wire#w5
   // the same network as SCL:
   "DB1723_UNIT_02_STA_3_ASPIRATION_VALVE"(OPTIONS_0 := 2#0000_0000,   // "FB1702_ASPIRATION_VALVE"
                           SWITCH_ON_CONDITIONS := "DB4000_FIX_TABLE_POSITIONS".UNIT_02.AXIS_E20_HOME_POS,
                           SWITCH_OFF_CONDITIONS := "DB7300_INTERLOCK_GENERAL".POWDER_PLC.FROM_POWDER_TO_UNIT_02.POWDER_UNIT_02_STOPPED OR "DB2120_MPP_ITC_IPC".STOP_SERVICES_GLOBAL,
                           HMI_LINE_REQUEST := "LTLP_DirectKeyGetMovNoData".Setup2[115],
                           SWITCH_ON_AUTO_REQUEST := NOT (NOT "DB362_M_UNIT_02_STA_3".M_CODES_UNIT_02_STA_3.M140 AND NOT "DB1101_MACHINE_SEQUENCE".RUNNING AND NOT "DB1251_PART_CYCLE_UNIT_02".RUNNING AND NOT "DB1255_UNIT_02_STATION_3_CYCLE".SEQUENCE.RUNNING),
                           SWITCH_OFF_AUTO_REQUEST := NOT (NOT "DB362_M_UNIT_02_STA_3".M_CODES_UNIT_02_STA_3.M141 AND NOT "DB2120_MPP_ITC_IPC".STOP_SERVICES_GLOBAL) OR (NOT "DB1101_MACHINE_SEQUENCE".RUNNING AND NOT "DB1251_PART_CYCLE_UNIT_02".RUNNING AND NOT "DB1255_UNIT_02_STATION_3_CYCLE".SEQUENCE.RUNNING),
                           SWITCH_OFF_GLOBAL_REQUEST := "DB7300_INTERLOCK_GENERAL".POWDER_PLC.FROM_POWDER_TO_UNIT_02.POWDER_UNIT_02_STOPPED AND "DB7300_INTERLOCK_GENERAL".POWDER_PLC.GENERAL.POWDER_PLC_AUTO_MODE,
                           UNIT_ALARM := 2,
                           STATION_ALARM := 3,
                           SIMULTANEITY_ALARM => "DB426_ALARMS_WARNINGS".SERVICES."709071",
                           TIME_EXCEEDED_ALARM => "DB426_ALARMS_WARNINGS".SERVICES."709072",
                           SWITCH_ON_ALARM => "DB426_ALARMS_WARNINGS".SERVICES."709073",
                           SWITCH_OFF_ALARM => "DB426_ALARMS_WARNINGS".SERVICES."709074",
                           HMI_MOTION_EXECUTABILITY_LEFT => "DB505_HMI_SetUp".Setup2.Movement_Executability.movement115ExecutabilityLeft,
                           HMI_MOTION_EXECUTABILITY_RIGHT => "DB505_HMI_SetUp".Setup2.Movement_Executability.movement115ExecutabilityRight,
                           HMI_MOTION_END_POS_LEFT => "DB505_HMI_SetUp".Setup2.Movement_EndPos.movement115EndPosLeft,
                           HMI_MOTION_END_POS_RIGHT => "DB505_HMI_SetUp".Setup2.Movement_EndPos.movement115EndPosRight,
                           HMI_MOTION_ACTIVE_LEFT => "DB505_HMI_SetUp".Setup2.MovementActive.movement115ActiveLeft,
                           HMI_MOTION_ACTIVE_RIGHT => "DB505_HMI_SetUp".Setup2.MovementActive.movement115ActiveRight,
                           SWITCH_ON => "Tag_13");
END_REGION

REGION Network 10: PRESSURE CONTROL STA 3 INPUT SENSOR VALUES
   RUNG wire#powerrail
      Contact( "M_ONE" )
      { S7_Templates := "[SrcType := Int, DestType := Real]" } Normalize(min := 0.0, value := "U02_STA_3_PRESSURE", max := 32240, out => "DB1799_ASPIRATION_AUX".UNIT_02_PRESSURE_CONTROL.STA_3_PRESSURE_CONTROL.NORMALIZED_VALUE)
      { S7_Templates := "[SrcType := Real, DestType := Real]" } Scale(min := -1000.0, value := "DB1799_ASPIRATION_AUX".UNIT_02_PRESSURE_CONTROL.STA_3_PRESSURE_CONTROL.NORMALIZED_VALUE, max := 1000.0, out => "DB1799_ASPIRATION_AUX".UNIT_02_PRESSURE_CONTROL.STA_3_PRESSURE_CONTROL.SCALED_VALUE)
      Move(in := "DB1799_ASPIRATION_AUX".UNIT_02_PRESSURE_CONTROL.STA_3_PRESSURE_CONTROL.SCALED_VALUE, out1 => "DB1799_ASPIRATION_AUX".UNIT_02_PRESSURE_CONTROL.STA_3_PRESSURE_CONTROL.FINAL_VALUE)
   END_RUNG
   // the same network as SCL:
   IF "M_ONE" THEN
       "DB1799_ASPIRATION_AUX".UNIT_02_PRESSURE_CONTROL.STA_3_PRESSURE_CONTROL.NORMALIZED_VALUE := NORM_X(MIN := 0.0, VALUE := "U02_STA_3_PRESSURE", MAX := 32240);
       "DB1799_ASPIRATION_AUX".UNIT_02_PRESSURE_CONTROL.STA_3_PRESSURE_CONTROL.SCALED_VALUE := SCALE_X(MIN := -1000.0, VALUE := "DB1799_ASPIRATION_AUX".UNIT_02_PRESSURE_CONTROL.STA_3_PRESSURE_CONTROL.NORMALIZED_VALUE, MAX := 1000.0);
       "DB1799_ASPIRATION_AUX".UNIT_02_PRESSURE_CONTROL.STA_3_PRESSURE_CONTROL.FINAL_VALUE := "DB1799_ASPIRATION_AUX".UNIT_02_PRESSURE_CONTROL.STA_3_PRESSURE_CONTROL.SCALED_VALUE;
   END_IF;
END_REGION

REGION Network 11: CALL FB1701 UNIT 02 STATION 4 ASPIRATION ACTIVATION
   // 2#0000_0001 OPTIONS 0 BIT 0 SWITCHED ON INPUT 1 OPTION
   // 2#0000_0010 OPTIONS 0 BIT 1 SWITCHED ON INPUT 2 OPTION
   // 2#0000_0100 OPTIONS 0 BIT 2 SWITCHED ON INPUT 3 OPTION
   // 2#0000_1000 OPTIONS 0 BIT 3 SWITCHED ON INPUT 4 OPTION
   // 2#0001_0000 OPTIONS 0 BIT 4 SWITCHED OFF NOT SWITCHED ON INPUT 1 OPTION
   // 2#0010_0000 OPTIONS 0 BIT 5 SPARE
   // 2#0100_0000 OPTIONS 0 BIT 6 SPARE
   // 2#1000_0000 OPTIONS 0 BIT 7 SPARE
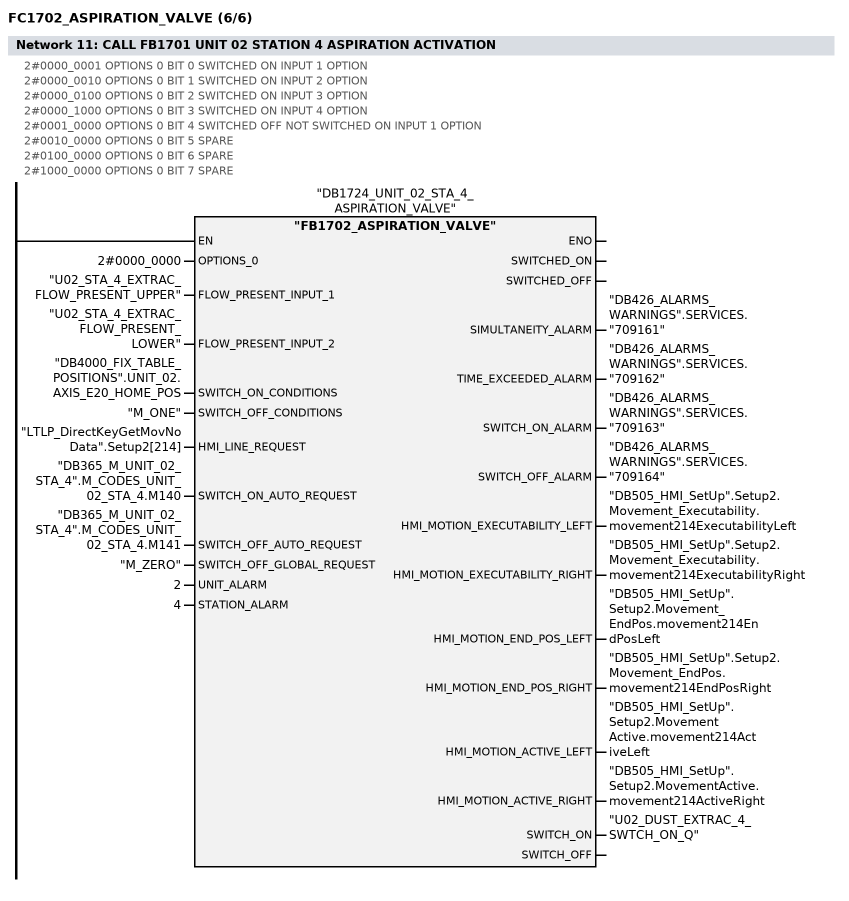
   RUNG wire#powerrail
      "DB1724_UNIT_02_STA_4_ASPIRATION_VALVE"(OPTIONS_0 := 2#0000_0000, FLOW_PRESENT_INPUT_1 := "U02_STA_4_EXTRAC_FLOW_PRESENT_UPPER", FLOW_PRESENT_INPUT_2 := "U02_STA_4_EXTRAC_FLOW_PRESENT_LOWER", SWITCH_ON_CONDITIONS := "DB4000_FIX_TABLE_POSITIONS".UNIT_02.AXIS_E20_HOME_POS, SWITCH_OFF_CONDITIONS := "M_ONE", HMI_LINE_REQUEST := "LTLP_DirectKeyGetMovNoData".Setup2[214], SWITCH_ON_AUTO_REQUEST := "DB365_M_UNIT_02_STA_4".M_CODES_UNIT_02_STA_4.M140, SWITCH_OFF_AUTO_REQUEST := "DB365_M_UNIT_02_STA_4".M_CODES_UNIT_02_STA_4.M141, SWITCH_OFF_GLOBAL_REQUEST := "M_ZERO", UNIT_ALARM := 2, STATION_ALARM := 4, SWITCHED_ON =>, SWITCHED_OFF =>, SIMULTANEITY_ALARM => "DB426_ALARMS_WARNINGS".SERVICES."709161", TIME_EXCEEDED_ALARM => "DB426_ALARMS_WARNINGS".SERVICES."709162", SWITCH_ON_ALARM => "DB426_ALARMS_WARNINGS".SERVICES."709163", SWITCH_OFF_ALARM => "DB426_ALARMS_WARNINGS".SERVICES."709164", HMI_MOTION_EXECUTABILITY_LEFT => "DB505_HMI_SetUp".Setup2.Movement_Executability.movement214ExecutabilityLeft, HMI_MOTION_EXECUTABILITY_RIGHT => "DB505_HMI_SetUp".Setup2.Movement_Executability.movement214ExecutabilityRight, HMI_MOTION_END_POS_LEFT => "DB505_HMI_SetUp".Setup2.Movement_EndPos.movement214EndPosLeft, HMI_MOTION_END_POS_RIGHT => "DB505_HMI_SetUp".Setup2.Movement_EndPos.movement214EndPosRight, HMI_MOTION_ACTIVE_LEFT => "DB505_HMI_SetUp".Setup2.MovementActive.movement214ActiveLeft, HMI_MOTION_ACTIVE_RIGHT => "DB505_HMI_SetUp".Setup2.MovementActive.movement214ActiveRight, SWITCH_ON => "U02_DUST_EXTRAC_4_SWTCH_ON_Q", SWITCH_OFF =>)
   END_RUNG
   // the same network as SCL:
   "DB1724_UNIT_02_STA_4_ASPIRATION_VALVE"(OPTIONS_0 := 2#0000_0000,   // "FB1702_ASPIRATION_VALVE"
                           FLOW_PRESENT_INPUT_1 := "U02_STA_4_EXTRAC_FLOW_PRESENT_UPPER",
                           FLOW_PRESENT_INPUT_2 := "U02_STA_4_EXTRAC_FLOW_PRESENT_LOWER",
                           SWITCH_ON_CONDITIONS := "DB4000_FIX_TABLE_POSITIONS".UNIT_02.AXIS_E20_HOME_POS,
                           SWITCH_OFF_CONDITIONS := "M_ONE",
                           HMI_LINE_REQUEST := "LTLP_DirectKeyGetMovNoData".Setup2[214],
                           SWITCH_ON_AUTO_REQUEST := "DB365_M_UNIT_02_STA_4".M_CODES_UNIT_02_STA_4.M140,
                           SWITCH_OFF_AUTO_REQUEST := "DB365_M_UNIT_02_STA_4".M_CODES_UNIT_02_STA_4.M141,
                           SWITCH_OFF_GLOBAL_REQUEST := "M_ZERO",
                           UNIT_ALARM := 2,
                           STATION_ALARM := 4,
                           SIMULTANEITY_ALARM => "DB426_ALARMS_WARNINGS".SERVICES."709161",
                           TIME_EXCEEDED_ALARM => "DB426_ALARMS_WARNINGS".SERVICES."709162",
                           SWITCH_ON_ALARM => "DB426_ALARMS_WARNINGS".SERVICES."709163",
                           SWITCH_OFF_ALARM => "DB426_ALARMS_WARNINGS".SERVICES."709164",
                           HMI_MOTION_EXECUTABILITY_LEFT => "DB505_HMI_SetUp".Setup2.Movement_Executability.movement214ExecutabilityLeft,
                           HMI_MOTION_EXECUTABILITY_RIGHT => "DB505_HMI_SetUp".Setup2.Movement_Executability.movement214ExecutabilityRight,
                           HMI_MOTION_END_POS_LEFT => "DB505_HMI_SetUp".Setup2.Movement_EndPos.movement214EndPosLeft,
                           HMI_MOTION_END_POS_RIGHT => "DB505_HMI_SetUp".Setup2.Movement_EndPos.movement214EndPosRight,
                           HMI_MOTION_ACTIVE_LEFT => "DB505_HMI_SetUp".Setup2.MovementActive.movement214ActiveLeft,
                           HMI_MOTION_ACTIVE_RIGHT => "DB505_HMI_SetUp".Setup2.MovementActive.movement214ActiveRight,
                           SWITCH_ON => "U02_DUST_EXTRAC_4_SWTCH_ON_Q");
END_REGION
END_FUNCTION
